PROGRAM MAIN
VAR
	{attribute addProperty Name "Horizontal piston A1"}
	_horizontalPiston : fbPneumaticActuator;
	{attribute addProperty Name "Vertical piston A2"}
	_verticalPiston : fbPneumaticActuator;
	{attribute addProperty Name "Gripper A3"}
	_gripper : fbPneumaticActuator;
	
END_VAR

_horizontalPiston.Manual();
_horizontalPiston.SimulateInputs();

_verticalPiston.Manual();
_verticalPiston.SimulateInputs();

_gripper.Manual();
_gripper.SimulateInputs();

END_PROGRAM

(* stored: Version 1.1.0.1, ProductVersion 3.1.4024.2
   POU MAIN: Id {16075815-a4a8-45db-abd4-3ff94277c648}, SpecialFunc None *)
